{attribute addProperty BoxType "EK1122-0000-0018"}
{attribute addProperty Id "Beckhoff_EQ2xxxsub_EK1100EK1100_179A0949162A_0001_EQ2008_0002_0016EQ2008_04E0E56B8811A_0002_EQ2008_0002_0017EQ2008_04E0E56B8811A_0003_EQ2008_0002_0018EQ2008_04E0E56B8811A_0004_EQ2008_0002_0019EQ2008_04E0E56B8811A_0005_EQ2339_0022_0016EQ2339_2F846F4A28836A_0006_EQ2339_0022_0017EQ2339_2F846F4A28836A_0007_EQ2339_0022_0018EQ2339_2F846F4A28836A_0008_EQ2339_0022_0019EQ2339_2F846F4A28836A_0009_EQ2809_0022_0016EQ2809_5A2A5F2915219A_0010_EQ2809_0022_0017EQ2809_5A2A5F2915219A_0011_EQ2809_0022_0018EQ2809_5A2A5F2915219"}
{attribute addProperty CRC "3922194899"}
{attribute addProperty SizeInBites "1976"}
{attribute addProperty SizeInBytes "247"}
TYPE Beckhoff_EQ2xxxEK1122_E9C7F1D3 EXTENDS EK1122_179A0949 :
STRUCT
	{attribute addProperty Name "Beckhoff_EQ2xxxsub_EK1100"}
	Beckhoff_EQ2xxxsub_EK1100 : EK1100_179A0949;
	{attribute addProperty Name "A_0001_EQ2008_0002_0016"}
	A_0001_EQ2008_0002_0016 : EQ2008_04E0E56B;
	{attribute addProperty Name "A_0002_EQ2008_0002_0017"}
	A_0002_EQ2008_0002_0017 : EQ2008_04E0E56B;
	{attribute addProperty Name "A_0003_EQ2008_0002_0018"}
	A_0003_EQ2008_0002_0018 : EQ2008_04E0E56B;
	{attribute addProperty Name "A_0004_EQ2008_0002_0019"}
	A_0004_EQ2008_0002_0019 : EQ2008_04E0E56B;
	{attribute addProperty Name "A_0005_EQ2339_0022_0016"}
	A_0005_EQ2339_0022_0016 : EQ2339_2F846F4A;
	{attribute addProperty Name "A_0006_EQ2339_0022_0017"}
	A_0006_EQ2339_0022_0017 : EQ2339_2F846F4A;
	{attribute addProperty Name "A_0007_EQ2339_0022_0018"}
	A_0007_EQ2339_0022_0018 : EQ2339_2F846F4A;
	{attribute addProperty Name "A_0008_EQ2339_0022_0019"}
	A_0008_EQ2339_0022_0019 : EQ2339_2F846F4A;
	{attribute addProperty Name "A_0009_EQ2809_0022_0016"}
	A_0009_EQ2809_0022_0016 : EQ2809_5A2A5F29;
	{attribute addProperty Name "A_0010_EQ2809_0022_0017"}
	A_0010_EQ2809_0022_0017 : EQ2809_5A2A5F29;
	{attribute addProperty Name "A_0011_EQ2809_0022_0018"}
	A_0011_EQ2809_0022_0018 : EQ2809_5A2A5F29;
END_STRUCT
END_TYPE

(* stored: Version 1.2.0.0, ProductVersion 3.1.4024.9
   DUT Beckhoff_EQ2xxxEK1122_E9C7F1D3: Id {d1b17a84-34bd-42a2-b531-cfb180725651} *)
